// TwinCAT 3 PLC project ConveyorPLC
// ProgramVersion: 3.1.4026.27
// libraries:
//   Tc2_Standard, * (Beckhoff Automation GmbH)
//   Tc2_System, * (Beckhoff Automation GmbH)
// project tree:
//   / PlcTask.TcTTO
//   POUs/ MAIN.TcPOU
// real-time tasks:
//   TASK PlcTask: cycle T#10ms, priority 20, ADS port 350
//   TASK PlcTask1: cycle T#10ms, priority 21, ADS port 351

CONFIGURATION ConveyorPLC
    RESOURCE PLC ON TwinCAT3
        TASK PlcTask(INTERVAL := T#10ms, PRIORITY := 21);
        PROGRAM MAIN WITH PlcTask : MAIN;
    END_RESOURCE
END_CONFIGURATION

// ---- POUs/MAIN.TcPOU
PROGRAM MAIN
VAR
	Lamp : BOOL;  //Lamp False is off True is on
	Timer : TON; // Lamp off Timer
	Timer2 : TON; //Lamp on Timer
END_VAR


//Turns the light on and off using two timers you can set them to be different times!
Timer(IN := NOT Lamp, PT := T#5000MS);
IF Timer.Q THEN
	Lamp := TRUE;
END_IF;

Timer2(IN := Lamp, PT := T#500MS);
IF Timer2.Q THEN
	Lamp := FALSE;
END_IF;


(*
//Toggles the light on and off on the same timer only uses 1 timer though.
Timer(IN := NOT Timer.Q,PT:= T#500MS);
IF Timer.Q THEN
	Lamp := NOT Lamp;
END_IF;

*)

END_PROGRAM
